(* IEC 61131-3 sources: Lasal/CPU_5344_V01/Class/cmBlower, 1 file *)

(* ---- cmBlower.st ---- *)
(*!
<Class
	Name               = "cmBlower"
	Revision           = "0.0"
	RealtimeTask       = "false"
	CyclicTask         = "true"
	DefCyclictime      = "10 ms"
	BackgroundTask     = "true"
	Sigmatek           = "false"
	OSInterface        = "false"
	HighPriority       = "false"
	Automatic          = "false"
	UpdateMode         = "Prescan"
	SharedCommandTable = "true"
	Objectsize         = "(450,1080)">
	<Channels>
		<Server Name="cmdBlow" Visualized="false" Initialize="false" WriteProtected="false" Retentive="false"/>
		<Server Name="parAmountOfBlows" Visualized="true" Initialize="true" DefValue="3" WriteProtected="false" Retentive="File"/>
		<Server Name="parTimeBlowOff" Visualized="true" Initialize="true" DefValue="500" WriteProtected="false" Retentive="File"/>
		<Server Name="parTimeBlowOn" Visualized="true" Initialize="true" DefValue="1000" WriteProtected="false" Retentive="File"/>
		<Server Name="stprBlow" Visualized="true" Initialize="false" WriteProtected="true" Retentive="false"/>
		<Server Name="stsCounter" Visualized="false" Initialize="false" WriteProtected="true" Retentive="false"/>
		<Client Name="oBlowValve" Required="false" Internal="false"/>
	</Channels>
	<Separators>
		<Servers>
			<SepChn Position="0"/>
			<SepChn Position="3"/>
			<SepChn Position="5"/>
		</Servers>
	</Separators>
	<Network Name="cmBlower">
		<!-- List of Components in this network -->
		<Components>
			<Object
				Name       = "_base"
				Class      = "cmBase"
				Position   = "(218,120)"
				Visualized = "true">
				<Channels>
					<Server Name="ClassSvr"/>
					<Server Name="cmdHMI"/>
					<Server Name="ErrorNr"/>
					<Server Name="mode"/>
					<Server Name="state"/>
					<Server Name="stsHMI_RunsAllowed"/>
					<Server Name="stsInAlarm"/>
					<Server Name="stsIsInterlocked"/>
					<Client Name="id"/>
					<Client Name="nwEmOrUnit"/>
				</Channels>
			</Object>
		</Components>
		<Comments>
		</Comments>
		<!-- List of Connections in this network -->
		<Connections>
			<Connection Source="this.ClassSvr" Destination="_base.ClassSvr" Vertices="(1036,210),(864,210),"/>
			<Connection Source="this.state" Destination="_base.state" Vertices="(1036,270),(864,270),"/>
			<Connection Source="this.mode" Destination="_base.mode" Vertices="(1036,330),(864,330),"/>
			<Connection Source="this.cmdHMI" Destination="_base.cmdHMI" Vertices="(1036,390),(864,390),"/>
			<Connection Source="this.stsInAlarm" Destination="_base.stsInAlarm" Vertices="(1036,450),(864,510),"/>
			<Connection Source="this.stsIsInterlocked" Destination="_base.stsIsInterlocked" Vertices="(1036,510),(864,570),"/>
			<Connection Source="this.stsHMI_RunsAllowed" Destination="_base.stsHMI_RunsAllowed" Vertices="(1036,570),(864,630),"/>
			<Connection Source="this.ErrorNr" Destination="_base.ErrorNr" Vertices="(1036,630),(864,690),"/>
			<Connection Source="_base.nwEmOrUnit" Destination="this.nwEmOrUnit" Vertices="(218,210),(38,210),"/>
			<Connection Source="_base.id" Destination="this.id" Vertices="(218,270),(38,270),"/>
		</Connections>
		<!-- Headerfiles -->
		<Options>
		</Options>
	</Network>
</Class>
*)
#pragma using cmBase

cmBlower : CLASS
: cmBase
  //Servers:
	stprBlow 	: SvrCh_DINT;
	stsCounter 	: SvrCh_DINT;
	cmdBlow 	: SvrCh_DINT;
	parTimeBlowOn 	: SvrCh_UDINT;
	parTimeBlowOff 	: SvrCh_UDINT;
	parAmountOfBlows 	: SvrCh_DINT;
  //Clients:
	oBlowValve 	: CltCh_DINT;
  //Variables:
		timerBlowOn 	: strTimer;
		timerBlowOf 	: strTimer;
  //Functions:

	FUNCTION VIRTUAL work;

	FUNCTION VIRTUAL execStart;

	FUNCTION VIRTUAL execStop;

	FUNCTION VIRTUAL preScanOverride;

	FUNCTION VIRTUAL postScanOverride;
  //Tables:
	FUNCTION @STD
		VAR_OUTPUT
			ret_code	: CONFSTATES;
		END_VAR;
	FUNCTION GLOBAL TAB @CT_;
END_CLASS;

// JdK 5-6-2019: cmBlower created for 4284/Traffiroad / standard MPS library
// function is to start blowing in pulses or not

FUNCTION VIRTUAL cmBlower::work

  CASE stprBlow OF

  0: //rest

  1: //set blower on
    oBlowValve:=1;
    IF timerBlowOn.done THEN
      stprBlow+=1;
    END_IF;

  2: //set blower off
    IF timerBlowOf.done THEN
      stsCounter+=1;
      stprBlow+=1;
    END_IF;

  3: //check if we should do it again, or we are done
    IF stsCounter < parAmountOfBlows THEN
      stprBlow:=1;
    ELSE
      stsCounter:= 0;
      stprBlow:=0;
    END_IF;

  END_CASE;

END_FUNCTION

FUNCTION VIRTUAL cmBlower::execStart

  stprBlow:=1; //start blowing cycle

END_FUNCTION

FUNCTION VIRTUAL cmBlower::execStop

  stprBlow:=0; //stop blowing

END_FUNCTION

FUNCTION VIRTUAL cmBlower::preScanOverride

  oBlowValve:=0; //set it to 0 every cycle, if we need it to one, it is written to 1 after prescan

  IF pmlCom.sts.isInterlocked THEN
    stprBlow:=0; //at interlock, stop with blowing
  END_IF;

  //start blowing if there is a command to blow
  IF cmdBlow= 1 & (pmlCom.sts.mode= auto | pmlCom.sts.mode= service) & stprBlow=0 THEN
    cmdBlow:= 0; //do command only once
    stsCounter:= 0;
    stprBlow:=1;
  END_IF;

  //run timers
  timerBlowOn:=runTimer(Active:=stprBlow=1, iMem:=timerBlowOn, TimerTime:=parTimeBlowOn, Pause:=FALSE);
  timerBlowOf:=runTimer(Active:=stprBlow=2, iMem:=timerBlowOf, TimerTime:=parTimeBlowOff, Pause:=FALSE);

END_FUNCTION

FUNCTION VIRTUAL cmBlower::postScanOverride

  oBlowValve.Write(input:=oBlowValve);

END_FUNCTION
